Staubli VAL3: refreshAction.pgx

program refreshAction(num x_nIndex, InstrItem& x_iAction[], num x_nDistance)
  local string l_sMessage
  local string l_sTitle
  local num i
  local string l_sAction
  local num l_nSize
begin
  //
  // INSTRUCTION
  //
  cls()
  // create a menu to edit the action
  call use:setSizeList(5,3,30,4)
  call use:setView(false)
  // show the title
  call tcp:getSize(l_nSize)
  call language:message(l_sMessage,124)
  l_sTitle=l_sMessage+toString("3",nIndexTool)+"/"+toString("",l_nSize-1)
  call tcp:getName(l_sMessage,nIndexTool)
  l_sTitle=l_sTitle+" "+l_sMessage
  call use:listcreate(l_sTitle)
  // get the action string
  call language:message(l_sMessage,176)
  // insert all the 3 action
  for i=0 to 2
    l_sAction=l_sMessage+toString("",i+1)+"> "+x_iAction[i].sType+" "+x_iAction[i].sData
    call use:listadd(l_sAction)
  endFor
  call language:message(l_sMessage,177)
  l_sMessage=l_sMessage+"> "+toString("",x_nDistance)+" mm"
  call use:listadd(l_sMessage)
  // show it
  call use:clear(0,13)
  call use:typeMenu(8,"OK")
  use:nView=x_nIndex
  call use:listupdate(0)
  //
end
